// TIA Portal V15.1 export
// export: Created 2026-01-09T13:45:14.1672711Z, ExportSetting WithDefaults, WithReadOnly, DisplayName Totally Integrated Automation Portal, DisplayVersion V15.1 Update 8, DisplayName TIA Portal Openness, DisplayVersion V15.1 Update 8, DisplayName STEP 7 Professional, DisplayVersion V15.1 Update 8, DisplayName WinCC Advanced, DisplayVersion V15.1 Update 8
FUNCTION_BLOCK "7.WEIGHT_PROCESS"   // FB7, LAD
{ S7_Optimized_Access := 'TRUE' }
VERSION : 0.1
// Chú ý:
// W_DU: nhập khối lượng giớ hạn dưới để tính SS_DUOI sai số dưới, ví dụ SV_IN cài là 1000kg, giới hạn dưới cài là W_DU=55kg, vì KL_BU=0.0 nên> SS_DUOI=1000-55=945kg
// W_RTD: cài đặt khối lượng rơi tự do, từ đó tính điểm cắt Rơi tự do, ví dụ W_RTD=95kg, khi đó điểm cắt Rơi tự do KL_RTD=1000-95=905kg
// Thực tế khi đó: cân sẽ được cân thô đến điểm cắt RTD là 905kg thì nó sẽ bắt đầu chuyển sang Cân Tinh,
// stored: AutoNumber false, CodeModifiedDate 2026-01-04T10:59:07.612582Z, CompileDate 2026-01-04T14:27:04.4561281Z, CreationDate 2024-10-12T12:36:08.0193576Z, DownloadWithoutReinit false, HandleErrorsWithinBlock false, InterfaceModifiedDate 2024-08-06T09:13:34.3012657Z, IsConsistent true, IsIECCheckEnabled false, IsKnowHowProtected false, IsRetainMemResEnabled false, IsWriteProtected false, LibraryConformanceStatus Warning: The object contains access to global data blocks., MemoryReserve 100, ModifiedDate 2026-01-04T11:31:32.9722655Z, ParameterModified 2024-08-06T08:53:48.4792275Z, PLCSimAdvancedSupport false, SetENOAutomatically False, StructureModified 2024-08-06T09:13:34.3012657Z, UDAEnableTagReadback false
   VAR_INPUT
      AUT : Bool;
      MAN1 : Bool;
      MAN2 : Bool;
      LOGIC : Bool;
      FAU : Bool;   // Tạm dừng cân trong mode Auto
      FU_IN : Bool;   // Nút nhấn báo đầy Silo (phần mềm ghi xuống)
      X_CLOCK : Bool;
      EMTY_IN : Bool;   // Nút nhấn (hoặc tín hiệu trên phần mềm) báo cân rỗng
      XNC_MAN : Bool;
      XNC_AUT : Bool;
      BU_TRU : Bool;   // Nếu =false thì CAN_DƯ luôn bằng 0
      SV_IN : Real;
      W_IN : Real;   // Khối lượng cân hiện tại
      W_RTD : Real;   // Khối lựng rơi tự do
      W_TR : Real;   // KL giới hạn trên
      W_DU : Real;   // KL giới hạn dưới
      T_ON : Real;   // Thời gian cân mở
      T_OFF : Real;   // Thời gian cân đóng
      T_DL : Real;   // Thời gian đợi rơi thêm
      SMT : Real;
      KL_Bu_Tru : Real;   // >0.0 là bù chủ động vào KL_BU, ngược lại sẽ dùng CAN DƯ
   END_VAR
   VAR_OUTPUT
      MAC_OUT : Real;
      PV_OUT : Real;
      PVA_OUT : Real;
      PVM_OUT : Real;
      FU_OUT : Bool;   // Báo cân đầy
      EM_OUT : Bool;
      W_OVER : Real;
      Q_OUT1 : Bool;
      Q_OUT2 : Bool;
      OVER : Bool;
      STA_RUN : Bool;
   END_VAR
   VAR RETAIN
      FU { ExternalAccessible := 'False'; ExternalVisible := 'False'; ExternalWritable := 'False'} : Bool;   // Bít nhớ báo cân đầy
      EM { ExternalAccessible := 'False'; ExternalVisible := 'False'; ExternalWritable := 'False'} : Bool;
      "CAN DU" { ExternalAccessible := 'False'; ExternalVisible := 'False'; ExternalWritable := 'False'} : Real;   // Nếu BU_TRU=false thì CAN_DU luôn =0
      PVA { ExternalAccessible := 'False'; ExternalVisible := 'False'; ExternalWritable := 'False'} : Real;
      PVM { ExternalAccessible := 'False'; ExternalVisible := 'False'; ExternalWritable := 'False'} : Real;
      TOFF { ExternalAccessible := 'False'; ExternalVisible := 'False'; ExternalWritable := 'False'} : Real;
      TON { ExternalAccessible := 'False'; ExternalVisible := 'False'; ExternalWritable := 'False'} : Real;
      T_DLFULL { ExternalAccessible := 'False'; ExternalVisible := 'False'; ExternalWritable := 'False'} : Real;   // Đếm thời gian báo đầy
      "T_DLT/T" { ExternalAccessible := 'False'; ExternalVisible := 'False'; ExternalWritable := 'False'} : Real;   // Đếm thời gian cho lượng rơi thêm
      KL_BU : Real;   // Nhập băng KL_tru_bu hoặc nếu cân bị Cân Dư
      CLK_DLE { ExternalAccessible := 'False'; ExternalVisible := 'False'; ExternalWritable := 'False'} : Bool;
      CLK_DLF { ExternalAccessible := 'False'; ExternalVisible := 'False'; ExternalWritable := 'False'} : Bool;
      "CLK_DLT/T" { ExternalAccessible := 'False'; ExternalVisible := 'False'; ExternalWritable := 'False'} : Bool;
      CLK_TT { ExternalAccessible := 'False'; ExternalVisible := 'False'; ExternalWritable := 'False'} : Bool;
      "TEMP_T/T" { ExternalAccessible := 'False'; ExternalVisible := 'False'; ExternalWritable := 'False'} : Bool;   // Hết thời gian đóng cân ==> mở cân
      "RUN_T/T" { ExternalAccessible := 'False'; ExternalVisible := 'False'; ExternalWritable := 'False'} : Bool;   // Bật chạy thô tinh sau khi hết thời gian đợi rơi thêm
   END_VAR
   VAR
      RUN_MAN : Bool;
      RUN_AUT : Bool;
      "CUA_T/T" : Bool;
      P_OUT1 : Bool;
      P_OUT2 : Bool;
      P_EMTY : Bool;
      P_FU : Bool;
   END_VAR
   VAR_TEMP
      "SS TREN" : Real;
      "SS DUOI" : Real;
      "KL RTD" : Real;   // Điểm cắt Rơi tự do
   END_VAR
   VAR_TEMP   // added for the SCL form of the ladder/FBD networks
      _w1 : Bool;
      _w2 : Bool;
      _w3 : Bool;
   END_VAR
BEGIN

REGION Network 1: MOVE MAC
   // Nếu BU_TRU=false thì CAN_Du luôn bằng 0, khi đó nếu KL_Bu_Tru không được nhập thì KL_BU luôn =0.0
   // Thực tế trong chưng trình này, các điều kiện đang khiến CAN_DU=0.0 và KL_BU=0.0
   // Khi đó SS_DUOI=SV_IN - W_DU
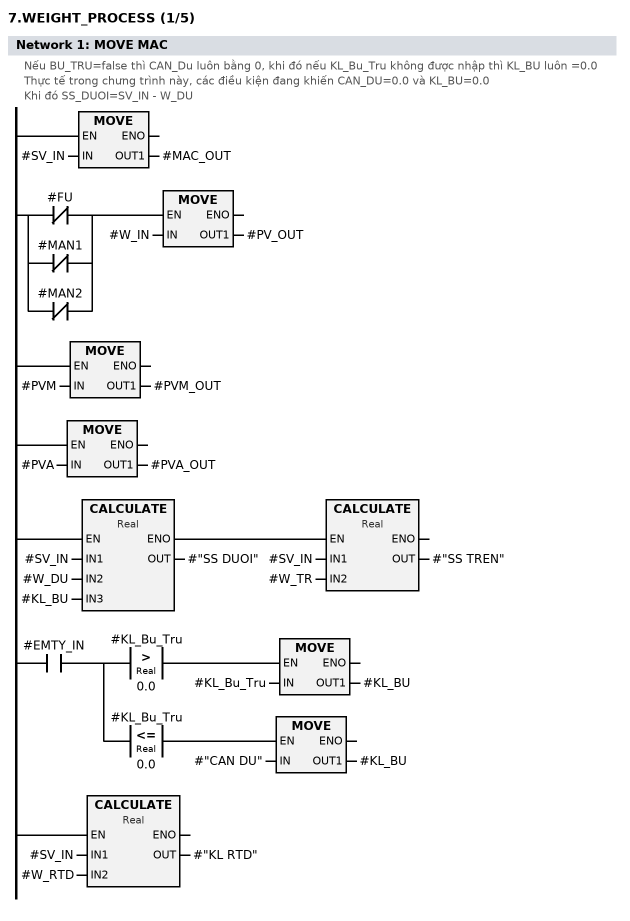
   RUNG wire#powerrail
      Move(in := #SV_IN, out1 => #MAC_OUT)
   END_RUNG
   RUNG wire#powerrail
      I_Contact( #FU )
      wire#w1
      Move(in := #W_IN, out1 => #PV_OUT)
   END_RUNG
   RUNG wire#powerrail
      I_Contact( #MAN1 )
   END_RUNG wire#w1
   RUNG wire#powerrail
      I_Contact( #MAN2 )
   END_RUNG wire#w1
   RUNG wire#powerrail
      Move(in := #PVM, out1 => #PVM_OUT)
   END_RUNG
   RUNG wire#powerrail
      Move(in := #PVA, out1 => #PVA_OUT)
   END_RUNG
   RUNG wire#powerrail
      { S7_Templates := "SrcType := Real"; S7_Expression := "IN1-IN2-IN3" } Calculate(in1 := #SV_IN, in2 := #W_DU, in3 := #KL_BU, out => #"SS DUOI")
      { S7_Templates := "SrcType := Real"; S7_Expression := "IN1+IN2" } Calculate(in1 := #SV_IN, in2 := #W_TR, out => #"SS TREN")
   END_RUNG
   RUNG wire#powerrail
      Contact( #EMTY_IN )
      wire#w2
      { S7_Templates := "SrcType := Real" } GT_Contact(in1 := #KL_Bu_Tru, in2 := 0.0)
      Move(in := #KL_Bu_Tru, out1 => #KL_BU)
   END_RUNG
   RUNG wire#w2
      { S7_Templates := "SrcType := Real" } LE_Contact(in1 := #KL_Bu_Tru, in2 := 0.0)
      Move(in := #"CAN DU", out1 => #KL_BU)
   END_RUNG
   RUNG wire#powerrail
      { S7_Templates := "SrcType := Real"; S7_Expression := "IN1-IN2" } Calculate(in1 := #SV_IN, in2 := #W_RTD, out => #"KL RTD")
   END_RUNG
   // the same network as SCL:
   #MAC_OUT := #SV_IN;
   IF NOT #FU OR NOT #MAN1 OR NOT #MAN2 THEN #PV_OUT := #W_IN; END_IF;
   #PVM_OUT := #PVM;
   #PVA_OUT := #PVA;
   #"SS DUOI" := #SV_IN-#W_DU-#KL_BU;
   #"SS TREN" := #SV_IN+#W_TR;
   IF #EMTY_IN AND (#KL_Bu_Tru > 0.0) THEN #KL_BU := #KL_Bu_Tru; END_IF;
   IF #EMTY_IN AND (#KL_Bu_Tru <= 0.0) THEN #KL_BU := #"CAN DU"; END_IF;
   #"KL RTD" := #SV_IN-#W_RTD;
END_REGION

REGION Network 2: KHOI LUONG CAN DU
   // Tính lượng CAN DƯ, khi cân FU, nếu vì lý do nào đó mà W_IN tiếp tục tăng, túc cân tiếp tục được nạp, thì  giá trị Dư đó xẽ được lưu lại vào biến #CAN DU
   // Báo tràn OVER: trong chế độ AUTO, nếu W_IN lớn hơn SS TRÊN sẽ báo tràn, khi bật FU_OUT thì không kích báo tràn tiếp được
   // Nhưng OVER này được giữ, nó chỉ bị reset khi xả cân, khi đó W_IN nhỏ hơn SS_TREN
   // W_OVER chính là lượng cân dư
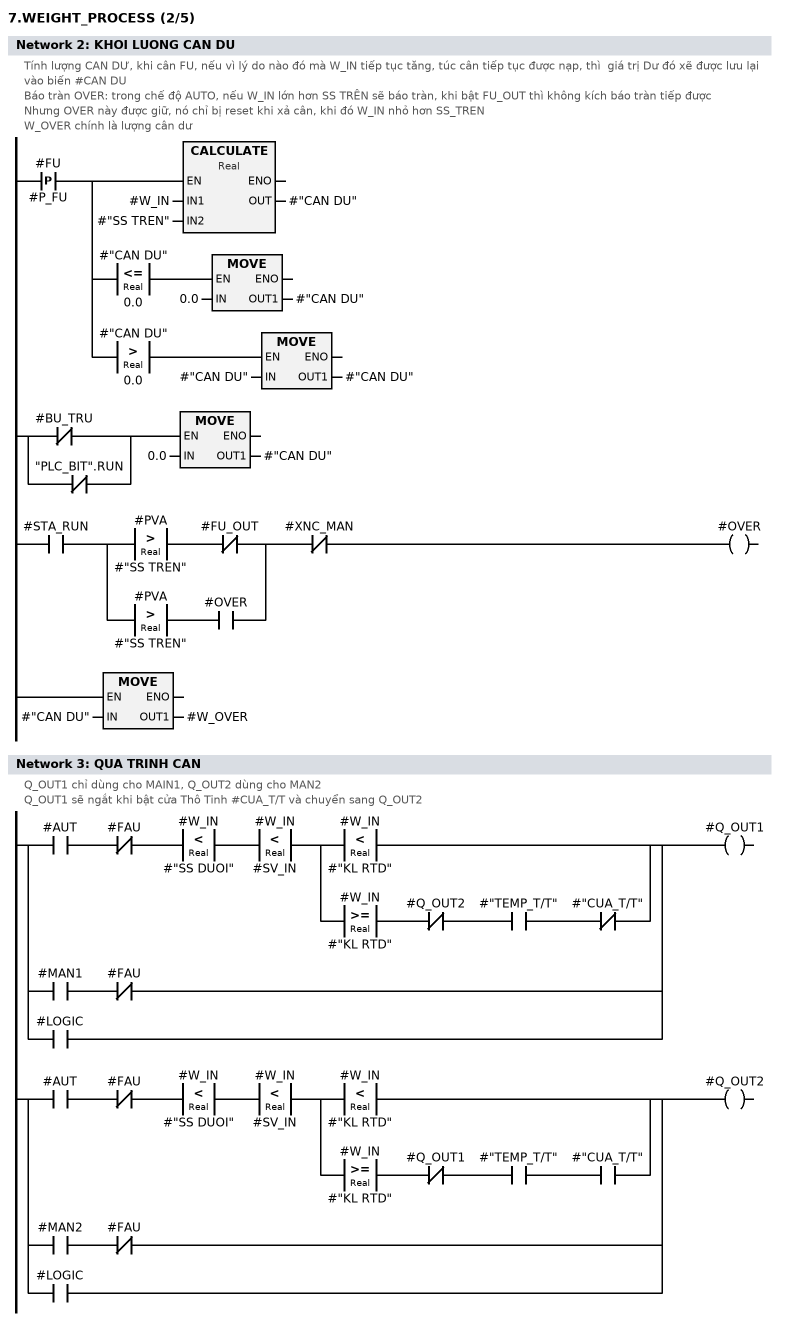
   RUNG wire#powerrail
      P_Contact(operand := #FU, bit := #P_FU)
      wire#w1
      { S7_Templates := "SrcType := Real"; S7_Expression := "IN1-IN2" } Calculate(in1 := #W_IN, in2 := #"SS TREN", out => #"CAN DU")
   END_RUNG
   RUNG wire#w1
      { S7_Templates := "SrcType := Real" } LE_Contact(in1 := #"CAN DU", in2 := 0.0)
      Move(in := 0.0, out1 => #"CAN DU")
   END_RUNG
   RUNG wire#w1
      { S7_Templates := "SrcType := Real" } GT_Contact(in1 := #"CAN DU", in2 := 0.0)
      Move(in := #"CAN DU", out1 => #"CAN DU")
   END_RUNG
   RUNG wire#powerrail
      I_Contact( #BU_TRU )
      wire#w2
      Move(in := 0.0, out1 => #"CAN DU")
   END_RUNG
   RUNG wire#powerrail
      I_Contact( "PLC_BIT".RUN )
   END_RUNG wire#w2
   RUNG wire#powerrail
      Contact( #STA_RUN )
      wire#w3
      { S7_Templates := "SrcType := Real" } GT_Contact(in1 := #PVA, in2 := #"SS TREN")
      I_Contact( #FU_OUT )
      wire#w4
      I_Contact( #XNC_MAN )
      Coil( #OVER )
   END_RUNG
   RUNG wire#w3
      { S7_Templates := "SrcType := Real" } GT_Contact(in1 := #PVA, in2 := #"SS TREN")
      Contact( #OVER )
   END_RUNG wire#w4
   RUNG wire#powerrail
      Move(in := #"CAN DU", out1 => #W_OVER)
   END_RUNG
   // the same network as SCL:
   #_w1 := #FU AND NOT #P_FU;   // rising edge of #FU
   #P_FU := #FU;
   IF #_w1 THEN #"CAN DU" := #W_IN-#"SS TREN"; END_IF;
   IF #_w1 AND (#"CAN DU" <= 0.0) THEN #"CAN DU" := 0.0; END_IF;
   IF #_w1 AND (#"CAN DU" > 0.0) THEN #"CAN DU" := #"CAN DU"; END_IF;
   IF NOT #BU_TRU OR NOT "PLC_BIT".RUN THEN #"CAN DU" := 0.0; END_IF;
   #OVER := #STA_RUN AND (((#PVA > #"SS TREN") AND NOT #FU_OUT) OR ((#PVA > #"SS TREN") AND #OVER)) AND NOT #XNC_MAN;
   #W_OVER := #"CAN DU";
END_REGION

REGION Network 3: QUA TRINH CAN
   // Q_OUT1 chỉ dùng cho MAIN1, Q_OUT2 dùng cho MAN2
   // Q_OUT1 sẽ ngắt khi bật cửa Thô Tinh #CUA_T/T và chuyển sang Q_OUT2
   RUNG wire#powerrail
      Contact( #AUT )
      I_Contact( #FAU )
      { S7_Templates := "SrcType := Real" } LT_Contact(in1 := #W_IN, in2 := #"SS DUOI")
      { S7_Templates := "SrcType := Real" } LT_Contact(in1 := #W_IN, in2 := #SV_IN)
      wire#w1
      { S7_Templates := "SrcType := Real" } LT_Contact(in1 := #W_IN, in2 := #"KL RTD")
      wire#w2
      Coil( #Q_OUT1 )
   END_RUNG
   RUNG wire#w1
      { S7_Templates := "SrcType := Real" } GE_Contact(in1 := #W_IN, in2 := #"KL RTD")
      I_Contact( #Q_OUT2 )
      Contact( #"TEMP_T/T" )
      I_Contact( #"CUA_T/T" )
   END_RUNG wire#w2
   RUNG wire#powerrail
      Contact( #MAN1 )
      I_Contact( #FAU )
   END_RUNG wire#w2
   RUNG wire#powerrail
      Contact( #LOGIC )
   END_RUNG wire#w2
   RUNG wire#powerrail
      Contact( #AUT )
      I_Contact( #FAU )
      { S7_Templates := "SrcType := Real" } LT_Contact(in1 := #W_IN, in2 := #"SS DUOI")
      { S7_Templates := "SrcType := Real" } LT_Contact(in1 := #W_IN, in2 := #SV_IN)
      wire#w3
      { S7_Templates := "SrcType := Real" } LT_Contact(in1 := #W_IN, in2 := #"KL RTD")
      wire#w4
      Coil( #Q_OUT2 )
   END_RUNG
   RUNG wire#w3
      { S7_Templates := "SrcType := Real" } GE_Contact(in1 := #W_IN, in2 := #"KL RTD")
      I_Contact( #Q_OUT1 )
      Contact( #"TEMP_T/T" )
      Contact( #"CUA_T/T" )
   END_RUNG wire#w4
   RUNG wire#powerrail
      Contact( #MAN2 )
      I_Contact( #FAU )
   END_RUNG wire#w4
   RUNG wire#powerrail
      Contact( #LOGIC )
   END_RUNG wire#w4
   // the same network as SCL:
   #Q_OUT1 := (#AUT AND NOT #FAU AND (#W_IN < #"SS DUOI") AND (#W_IN < #SV_IN) AND ((#W_IN < #"KL RTD") OR ((#W_IN >= #"KL RTD") AND NOT #Q_OUT2 AND #"TEMP_T/T" AND NOT #"CUA_T/T"))) OR (#MAN1 AND NOT #FAU) OR #LOGIC;
   #Q_OUT2 := (#AUT AND NOT #FAU AND (#W_IN < #"SS DUOI") AND (#W_IN < #SV_IN) AND ((#W_IN < #"KL RTD") OR ((#W_IN >= #"KL RTD") AND NOT #Q_OUT1 AND #"TEMP_T/T" AND #"CUA_T/T"))) OR (#MAN2 AND NOT #FAU) OR #LOGIC;
END_REGION

REGION Network 4: CHIA PV
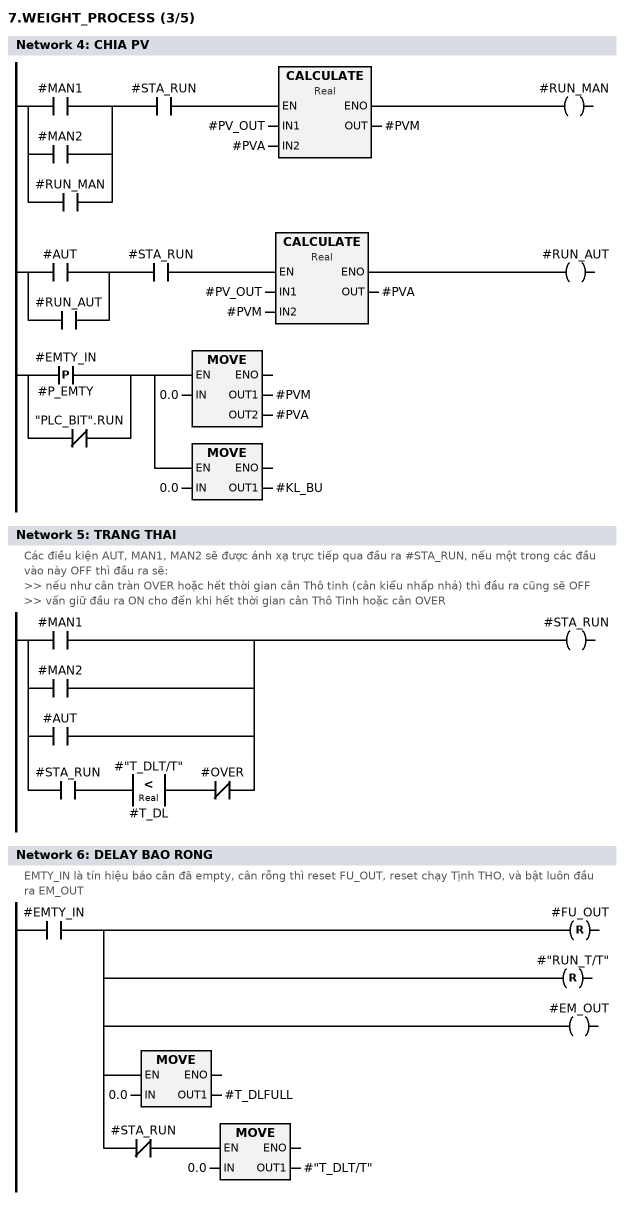
   RUNG wire#powerrail
      Contact( #MAN1 )
      wire#w1
      Contact( #STA_RUN )
      { S7_Templates := "SrcType := Real"; S7_Expression := "IN1-IN2" } Calculate(in1 := #PV_OUT, in2 := #PVA, out => #PVM)
      Coil( #RUN_MAN )
   END_RUNG
   RUNG wire#powerrail
      Contact( #MAN2 )
   END_RUNG wire#w1
   RUNG wire#powerrail
      Contact( #RUN_MAN )
   END_RUNG wire#w1
   RUNG wire#powerrail
      Contact( #AUT )
      wire#w2
      Contact( #STA_RUN )
      { S7_Templates := "SrcType := Real"; S7_Expression := "IN1-IN2" } Calculate(in1 := #PV_OUT, in2 := #PVM, out => #PVA)
      Coil( #RUN_AUT )
   END_RUNG
   RUNG wire#powerrail
      Contact( #RUN_AUT )
   END_RUNG wire#w2
   RUNG wire#powerrail
      P_Contact(operand := #EMTY_IN, bit := #P_EMTY)
      wire#w3
      Move(in := 0.0, out1 => #PVM, out2 => #PVA)
   END_RUNG
   RUNG wire#powerrail
      I_Contact( "PLC_BIT".RUN )
   END_RUNG wire#w3
   RUNG wire#w3
      Move(in := 0.0, out1 => #KL_BU)
   END_RUNG
   // the same network as SCL:
   #_w1 := (#MAN1 OR #MAN2 OR #RUN_MAN) AND #STA_RUN;
   IF #_w1 THEN #PVM := #PV_OUT-#PVA; END_IF;
   #RUN_MAN := #_w1;
   #_w2 := (#AUT OR #RUN_AUT) AND #STA_RUN;
   IF #_w2 THEN #PVA := #PV_OUT-#PVM; END_IF;
   #RUN_AUT := #_w2;
   #_w3 := #EMTY_IN AND NOT #P_EMTY;   // rising edge of #EMTY_IN
   #P_EMTY := #EMTY_IN;
   IF #_w3 OR NOT "PLC_BIT".RUN THEN
       #PVM := 0.0;
       #PVA := 0.0;
       #KL_BU := 0.0;
   END_IF;
END_REGION

REGION Network 5: TRANG THAI
   // Các điều kiện AUT, MAN1, MAN2 sẽ được ánh xạ trực tiếp qua đầu ra #STA_RUN, nếu một trong các đầu vào này OFF thì đầu ra sẽ:
   // >> nếu như cân tràn OVER hoặc hết thời gian cân Thô tinh (cân kiểu nhấp nhả) thì đầu ra cũng sẽ OFF
   // >> vấn giữ đầu ra ON cho đến khi hết thời gian cân Thô Tinh hoặc cân OVER
   RUNG wire#powerrail
      Contact( #MAN1 )
      wire#w1
      Coil( #STA_RUN )
   END_RUNG
   RUNG wire#powerrail
      Contact( #MAN2 )
   END_RUNG wire#w1
   RUNG wire#powerrail
      Contact( #AUT )
   END_RUNG wire#w1
   RUNG wire#powerrail
      Contact( #STA_RUN )
      { S7_Templates := "SrcType := Real" } LT_Contact(in1 := #"T_DLT/T", in2 := #T_DL)
      I_Contact( #OVER )
   END_RUNG wire#w1
   // the same network as SCL:
   #STA_RUN := #MAN1 OR #MAN2 OR #AUT OR (#STA_RUN AND (#"T_DLT/T" < #T_DL) AND NOT #OVER);
END_REGION

REGION Network 6: DELAY BAO RONG
   // EMTY_IN là tín hiệu báo cân đã empty, cân rỗng thì reset FU_OUT, reset chạy Tịnh THO, và bật luôn đầu ra EM_OUT
   RUNG wire#powerrail
      Contact( #EMTY_IN )
      wire#w1
      R_Coil( #FU_OUT )
   END_RUNG
   RUNG wire#w1
      R_Coil( #"RUN_T/T" )
   END_RUNG
   RUNG wire#w1
      Coil( #EM_OUT )
   END_RUNG
   RUNG wire#w1
      Move(in := 0.0, out1 => #T_DLFULL)
   END_RUNG
   RUNG wire#w1
      I_Contact( #STA_RUN )
      Move(in := 0.0, out1 => #"T_DLT/T")
   END_RUNG
   // the same network as SCL:
   IF #EMTY_IN THEN
       #FU_OUT := FALSE;
       #"RUN_T/T" := FALSE;
   END_IF;
   #EM_OUT := #EMTY_IN;
   IF #EMTY_IN THEN #T_DLFULL := 0.0; END_IF;
   IF #EMTY_IN AND NOT #STA_RUN THEN #"T_DLT/T" := 0.0; END_IF;
END_REGION

REGION Network 7: DELAY BAO DAY
   // Khi khối lượng đầu vào vượt qua sai số dưới, thì bắt đầu đếm để tình thời gian Delay trước khi báo FU
   // nếu thời gian đếm nó vượt qua giá trị cài đặt (cũng chính là thời gian đợi chơ lượng rơi thêm), thì SET ngõ ra #FU_OUT
   // 
   // Chú ý: chế độ MAN thì nó không báo FU
   // Cân FULL khi giá trị cân nó vượt qua SS_DUOI rồi đợi thêm một khoảng thời gian rơi thêm
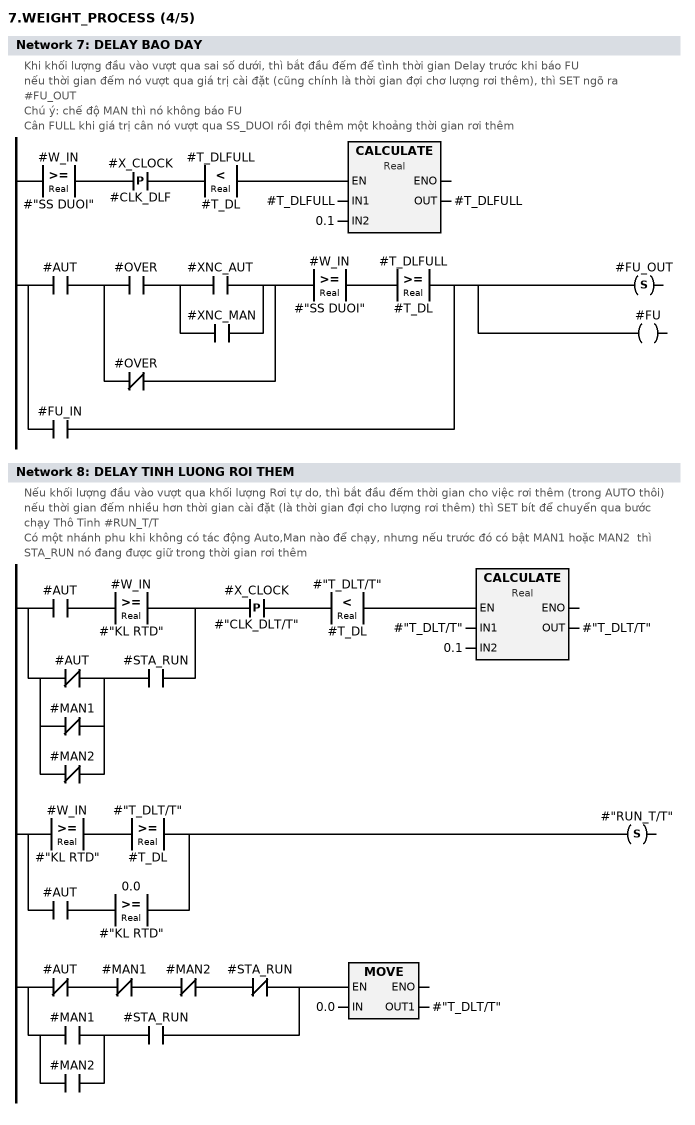
   RUNG wire#powerrail
      { S7_Templates := "SrcType := Real" } GE_Contact(in1 := #W_IN, in2 := #"SS DUOI")
      P_Contact(operand := #X_CLOCK, bit := #CLK_DLF)
      { S7_Templates := "SrcType := Real" } LT_Contact(in1 := #T_DLFULL, in2 := #T_DL)
      { S7_Templates := "SrcType := Real"; S7_Expression := "IN1+IN2" } Calculate(in1 := #T_DLFULL, in2 := 0.1, out => #T_DLFULL)
   END_RUNG
   RUNG wire#powerrail
      Contact( #AUT )
      wire#w1
      Contact( #OVER )
      wire#w2
      Contact( #XNC_AUT )
      wire#w3
      { S7_Templates := "SrcType := Real" } GE_Contact(in1 := #W_IN, in2 := #"SS DUOI")
      { S7_Templates := "SrcType := Real" } GE_Contact(in1 := #T_DLFULL, in2 := #T_DL)
      wire#w4
      S_Coil( #FU_OUT )
   END_RUNG
   RUNG wire#w2
      Contact( #XNC_MAN )
   END_RUNG wire#w3
   RUNG wire#w1
      I_Contact( #OVER )
   END_RUNG wire#w3
   RUNG wire#powerrail
      Contact( #FU_IN )
   END_RUNG wire#w4
   RUNG wire#w4
      Coil( #FU )
   END_RUNG
   // the same network as SCL:
   #_w1 := (#W_IN >= #"SS DUOI") AND #X_CLOCK AND NOT #CLK_DLF;   // rising edge of #X_CLOCK
   #CLK_DLF := #X_CLOCK;
   IF #_w1 AND (#T_DLFULL < #T_DL) THEN #T_DLFULL := #T_DLFULL+0.1; END_IF;
   #_w2 := (#AUT AND ((#OVER AND (#XNC_AUT OR #XNC_MAN)) OR NOT #OVER) AND (#W_IN >= #"SS DUOI") AND (#T_DLFULL >= #T_DL)) OR #FU_IN;
   IF #_w2 THEN #FU_OUT := TRUE; END_IF;
   #FU := #_w2;
END_REGION

REGION Network 8: DELAY TINH LUONG ROI THEM
   // Nếu khối lượng đầu vào vượt qua khối lượng Rơi tự do, thì bắt đầu đếm thời gian cho việc rơi thêm (trong AUTO thôi)
   // nếu thời gian đếm nhiều hơn thời gian cài đặt (là thời gian đợi cho lượng rơi thêm) thì SET bít để chuyển qua bước chạy Thô Tinh #RUN_T/T
   // 
   // Có một nhánh phu khi không có tác động Auto,Man nào để chạy, nhưng nếu trước đó có bật MAN1 hoặc MAN2  thì STA_RUN nó đang được giữ trong thời gian rơi thêm
   RUNG wire#powerrail
      Contact( #AUT )
      { S7_Templates := "SrcType := Real" } GE_Contact(in1 := #W_IN, in2 := #"KL RTD")
      wire#w1
      P_Contact(operand := #X_CLOCK, bit := #"CLK_DLT/T")
      { S7_Templates := "SrcType := Real" } LT_Contact(in1 := #"T_DLT/T", in2 := #T_DL)
      { S7_Templates := "SrcType := Real"; S7_Expression := "IN1+IN2" } Calculate(in1 := #"T_DLT/T", in2 := 0.1, out => #"T_DLT/T")
   END_RUNG
   RUNG wire#powerrail
      I_Contact( #AUT )
      wire#w2
      Contact( #STA_RUN )
   END_RUNG wire#w1
   RUNG wire#powerrail
      I_Contact( #MAN1 )
   END_RUNG wire#w2
   RUNG wire#powerrail
      I_Contact( #MAN2 )
   END_RUNG wire#w2
   RUNG wire#powerrail
      { S7_Templates := "SrcType := Real" } GE_Contact(in1 := #W_IN, in2 := #"KL RTD")
      { S7_Templates := "SrcType := Real" } GE_Contact(in1 := #"T_DLT/T", in2 := #T_DL)
      wire#w3
      S_Coil( #"RUN_T/T" )
   END_RUNG
   RUNG wire#powerrail
      Contact( #AUT )
      { S7_Templates := "SrcType := Real" } GE_Contact(in1 := 0.0, in2 := #"KL RTD")
   END_RUNG wire#w3
   RUNG wire#powerrail
      I_Contact( #AUT )
      I_Contact( #MAN1 )
      I_Contact( #MAN2 )
      I_Contact( #STA_RUN )
      wire#w4
      Move(in := 0.0, out1 => #"T_DLT/T")
   END_RUNG
   RUNG wire#powerrail
      Contact( #MAN1 )
      wire#w5
      Contact( #STA_RUN )
   END_RUNG wire#w4
   RUNG wire#powerrail
      Contact( #MAN2 )
   END_RUNG wire#w5
   // the same network as SCL:
   #_w1 := ((#AUT AND (#W_IN >= #"KL RTD")) OR ((NOT #AUT OR NOT #MAN1 OR NOT #MAN2) AND #STA_RUN)) AND #X_CLOCK AND NOT #"CLK_DLT/T";   // rising edge of #X_CLOCK
   #"CLK_DLT/T" := #X_CLOCK;
   IF #_w1 AND (#"T_DLT/T" < #T_DL) THEN #"T_DLT/T" := #"T_DLT/T"+0.1; END_IF;
   IF ((#W_IN >= #"KL RTD") AND (#"T_DLT/T" >= #T_DL)) OR (#AUT AND (0.0 >= #"KL RTD")) THEN
       #"RUN_T/T" := TRUE;
   END_IF;
   IF (NOT #AUT AND NOT #MAN1 AND NOT #MAN2 AND NOT #STA_RUN) OR ((#MAN1 OR #MAN2) AND #STA_RUN) THEN
       #"T_DLT/T" := 0.0;
   END_IF;
END_REGION

REGION Network 9: CAN THO TINH
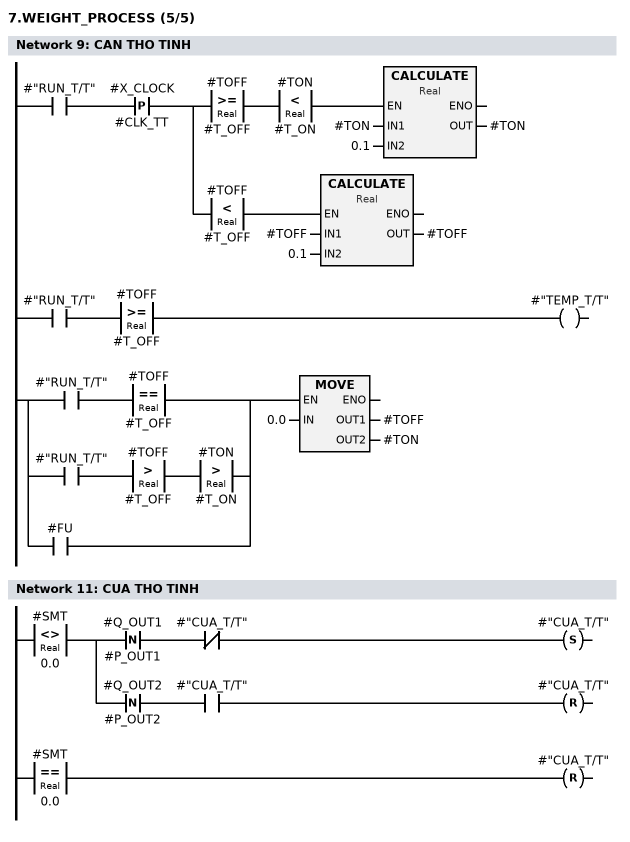
   RUNG wire#powerrail
      Contact( #"RUN_T/T" )
      P_Contact(operand := #X_CLOCK, bit := #CLK_TT)
      wire#w1
      { S7_Templates := "SrcType := Real" } GE_Contact(in1 := #TOFF, in2 := #T_OFF)
      { S7_Templates := "SrcType := Real" } LT_Contact(in1 := #TON, in2 := #T_ON)
      { S7_Templates := "SrcType := Real"; S7_Expression := "IN1+IN2" } Calculate(in1 := #TON, in2 := 0.1, out => #TON)
   END_RUNG
   RUNG wire#w1
      { S7_Templates := "SrcType := Real" } LT_Contact(in1 := #TOFF, in2 := #T_OFF)
      { S7_Templates := "SrcType := Real"; S7_Expression := "IN1+IN2" } Calculate(in1 := #TOFF, in2 := 0.1, out => #TOFF)
   END_RUNG
   RUNG wire#powerrail
      Contact( #"RUN_T/T" )
      { S7_Templates := "SrcType := Real" } GE_Contact(in1 := #TOFF, in2 := #T_OFF)
      Coil( #"TEMP_T/T" )
   END_RUNG
   RUNG wire#powerrail
      Contact( #"RUN_T/T" )
      { S7_Templates := "SrcType := Real" } EQ_Contact(in1 := #TOFF, in2 := #T_OFF)
      wire#w2
      Move(in := 0.0, out1 => #TOFF, out2 => #TON)
   END_RUNG
   RUNG wire#powerrail
      Contact( #"RUN_T/T" )
      { S7_Templates := "SrcType := Real" } GT_Contact(in1 := #TOFF, in2 := #T_OFF)
      { S7_Templates := "SrcType := Real" } GT_Contact(in1 := #TON, in2 := #T_ON)
   END_RUNG wire#w2
   RUNG wire#powerrail
      Contact( #FU )
   END_RUNG wire#w2
   // the same network as SCL:
   #_w1 := #"RUN_T/T" AND #X_CLOCK AND NOT #CLK_TT;   // rising edge of #X_CLOCK
   #CLK_TT := #X_CLOCK;
   IF #_w1 AND (#TOFF >= #T_OFF) AND (#TON < #T_ON) THEN #TON := #TON+0.1; END_IF;
   IF #_w1 AND (#TOFF < #T_OFF) THEN #TOFF := #TOFF+0.1; END_IF;
   #"TEMP_T/T" := #"RUN_T/T" AND (#TOFF >= #T_OFF);
   IF (#"RUN_T/T" AND (#TOFF = #T_OFF)) OR (#"RUN_T/T" AND (#TOFF > #T_OFF) AND (#TON > #T_ON)) OR #FU THEN
       #TOFF := 0.0;
       #TON := 0.0;
   END_IF;
END_REGION

REGION Network 10: CAN LOGIC
END_REGION

REGION Network 11: CUA THO TINH
   RUNG wire#powerrail
      { S7_Templates := "SrcType := Real" } NE_Contact(in1 := #SMT, in2 := 0.0)
      wire#w1
      N_Contact(operand := #Q_OUT1, bit := #P_OUT1)
      I_Contact( #"CUA_T/T" )
      S_Coil( #"CUA_T/T" )
   END_RUNG
   RUNG wire#w1
      N_Contact(operand := #Q_OUT2, bit := #P_OUT2)
      Contact( #"CUA_T/T" )
      R_Coil( #"CUA_T/T" )
   END_RUNG
   RUNG wire#powerrail
      { S7_Templates := "SrcType := Real" } EQ_Contact(in1 := #SMT, in2 := 0.0)
      R_Coil( #"CUA_T/T" )
   END_RUNG
   // the same network as SCL:
   #_w1 := #SMT <> 0.0;
   #_w2 := #_w1 AND NOT #Q_OUT1 AND #P_OUT1;   // falling edge of #Q_OUT1
   #P_OUT1 := #Q_OUT1;
   IF #_w2 AND NOT #"CUA_T/T" THEN #"CUA_T/T" := TRUE; END_IF;
   #_w3 := #_w1 AND NOT #Q_OUT2 AND #P_OUT2;   // falling edge of #Q_OUT2
   #P_OUT2 := #Q_OUT2;
   IF #_w3 AND #"CUA_T/T" THEN #"CUA_T/T" := FALSE; END_IF;
   IF #SMT = 0.0 THEN #"CUA_T/T" := FALSE; END_IF;
END_REGION
END_FUNCTION_BLOCK
